(* CoDeSys 2.3 library: cul_plc.lib *)

(* Global variable list: Globale_Variablen *)
VAR_GLOBAL CONSTANT
	Cul_PLC_LIBVER:				STRING(16) := 'V1.01 Release';	(* Version String *)
    Cul_PLC_MMPREADY:           BOOL       := TRUE;         (* MMP Ready *)

	(* Error return values *)
	Cul_ERC_Other:              DINT := -1;     (* CAN-function unsuccessful *)
    Cul_ERC_ParmInvalid:        DINT := -2;     (* parameters are invalid *)
	Cul_ERC_NoObj:              DINT := -3;     (* card/network not found/existing *)
	Cul_ERC_NoMemory :          DINT := -10;    (* Memory- or Thread-Alloc-Fail *)
END_VAR

(* POU CUL_AttachEvent, ST *)
(******************************************************************************
Description: attach/detach application events. 
Input:
	- Req:      request enable
	- NetNb:    1..8 Netnumber, attach event 
                (-1  show events, -2  detach events)
	- Event:    0  all flags (0x1f0000)
                16#04000xxx  Message
                16#0c000xxx  Message exclusive
                16#0400ffff  All Message
                16#0c00ffff  All Message exclusive
                16#1c00ffff  All existing Message exclusive
Output:
    - NbOfEvents:   Number of event-sessions started
    - Done:         TRUE means completed
    - Error:        TRUE in case of error
    - Status:       0: OK/Done, 1: BUSY, error-number in case of error
                    Cul_ERC_Other    error at/detaching event(s)
                    Cul_ERC_NoObj    network not found
******************************************************************************)
FUNCTION_BLOCK CUL_AttachEvent
VAR_INPUT
	Req : BOOL;
	NetNb: DINT;
END_VAR
VAR_IN_OUT
	Event: UDINT;
END_VAR
VAR_OUTPUT
	NbOfEvents: UDINT;
	Done : BOOL;
	Error : BOOL;
	Status : DINT;
END_VAR
VAR
	Pltd: DWORD;
END_VAR
;
END_FUNCTION_BLOCK

(* POU Cul_DetachEvent, ST *)
(******************************************************************************
Description: attach/detach application events of a net. 
Input:
	- NetNb:    1..8 Netnumber
	- Event:    0    all events
                <> 0 specific event

Return: 
	- >=0             number of detaches done
    - Cul_ERC_NoObj   net not found
******************************************************************************)
FUNCTION Cul_DetachEvent : DINT
VAR_INPUT
	NetNb: DINT;
    Event: UDINT;
END_VAR
VAR
END_VAR
;
END_FUNCTION

(* POU Cul_EnableMsg, ST *)
(******************************************************************************
Description: enable the receiption of a specific CAN-message by its COB-ID
Input:
	- CardNb:   Number of the card
    - Chan:     0 = CAN A, 1 = CAN B
	- CobId:    0..7ff  COB-ID of the CAN-Message which should be enabled for 
                receiption
Return: 
	- 0               Ok (message will be queued into the Rx-Queue)
    - Cul_ERC_NoObj   card not found or invalid COB-ID
******************************************************************************)
FUNCTION Cul_EnableMsg : DINT
VAR_INPUT
	CardNb: DINT;
	Chan: UDINT;
	CobId: UDINT;
END_VAR
VAR
END_VAR
;
END_FUNCTION

(* POU Cul_GetVersion, ST *)
(******************************************************************************
Description: Returns the version string of the library. In simulation always
	'V1.00 Release' is returned.

Input:
	- dummy

Return: 
	Version String
******************************************************************************)
FUNCTION Cul_GetVersion : STRING(15)
VAR_INPUT
	dummy :	BOOL;
END_VAR
VAR
END_VAR
cul_GetVersion := 'V1.00 Release';
END_FUNCTION

(* POU CUL_ReceiveMsg, ST *)
(******************************************************************************
Description: receive a message from the CAN-bus
             (get a message from the receive-queue). 
Input: 
    - NetNb:       1..8 Netnumber, attach event 
Output:
	- Event:       attached event
    - CobId:       COB-ID of the CAN-message
    - Rtr:         RTR of the CAN-message
    - Msg_Data:    receive data buffer
	- Msg_Length:  length of received message
    - Msg_Left:    number of messages still queued in the receive-queue
    - Status:      0   Ok
                   Cul_ERC_NoObj   no message in the receive-queue
******************************************************************************)
FUNCTION_BLOCK CUL_ReceiveMsg
VAR_INPUT
	NetNb: DINT;
END_VAR
VAR_OUTPUT
	Event: UDINT;
	CobId: UDINT;
	Rtr: UINT;
	Msg_Data : ARRAY [0..7] OF BYTE;
	Msg_Length : USINT;
	Msg_Left : USINT;
	Status : DINT;
END_VAR
VAR
END_VAR
;
END_FUNCTION_BLOCK

(* POU Cul_SendMsg, ST *)
(******************************************************************************
Description: send a message over the CAN-bus, 
             can block runtime. 

	NetNb:       1..8     CAN netnumber
	CobId:       0..7ff   COB-ID of the CAN-message
	Msg_Length:  0..8 | 0x10  data length or RTR
    Msg_Data:    data to transmit
Return: 
  	- 0                Ok
	- Cul_ERC_NoObj    net not found
******************************************************************************)
FUNCTION Cul_SendMsg : DINT
VAR_INPUT
	NetNb: DINT;
	CobId: UDINT;
	Msg_Data: ARRAY[0..7] OF BYTE;
	Msg_Length: USINT;
END_VAR
VAR
END_VAR
;
END_FUNCTION

(* POU CUL_SendMsg_NB, ST *)
(******************************************************************************
	Description: send a message over the CAN-bus, 
                 does not block the runtime. 

	Req:         request enable
	NetNb:       1..8     CAN netnumber
	CobId:       0..7ff   COB-ID of the CAN-message
	Msg_Length:  0..8 | 0x10  data length or RTR
    Msg_Data:    data to transmit
Return: 
    - Done:         TRUE means completed
    - Error:        TRUE in case of error
    - Status:       0: OK/Done, 1: BUSY, error-number in case of error
                    Cul_ERC_NoObj    network not found
******************************************************************************)
FUNCTION_BLOCK CUL_SendMsg_NB
VAR_INPUT
	Req: BOOL;
	NetNb: DINT;
	CobId: UDINT;
	Msg_Data: ARRAY[0..7] OF BYTE;
	Msg_Length: USINT;
END_VAR
VAR_OUTPUT
	Done: BOOL;
	Error: BOOL;
	Status: DINT;
END_VAR
VAR
	Pltd: DWORD;
END_VAR
;
END_FUNCTION_BLOCK
